Staubli VAL3: AfterCloseLaser.pgx

public program AfterCloseLaser(num x_nWorkplaceIn, num x_nTrajIndex)
begin
  //参数：x_nWorkplaceIn 工位序号，传入的参数是 DataBase:nWorkPlaceIndex
  //参数：x_nTrajIndex 路径序号，传入的参数是TxtFile:nReadTrajIndex
  //引用位置:Motion:Move.pgx
  //功能：激光关闭以后需要做的动作
  //备注：离开点还没有运行之前




end
